// Mitsubishi GX Works2 project: Group 7 PLC   PLC: FX3G

// global labels: Global1
VAR_GLOBAL
  Emergency AT X005 : BOOL;
  PowerButton AT X007 : BOOL;
  PowerOn AT Y007 : BOOL;
  analog_input_1 AT D8280 : INT;
END_VAR
VAR_GLOBAL CONSTANT
  div_analog : REAL := 400.0;
  max_regular : REAL := 5.0;
  min_pinuk : REAL := 6.0;
END_VAR
VAR_GLOBAL
  pinuk AT M1 : BOOL;  (* fictive lamp that represent pinuk choise *)
  regular AT M2 : BOOL;  (* fictive lamp that represent regular choise *)
  RaspberryInput AT D1100 : REAL;
  LemonInput AT D1102 : REAL;
  StabilizerInput AT D1104 : REAL;
  GummyBearInput AT D1106 : REAL;
  RaspberryStock AT D1108 : REAL;
  LemonStock AT D1110 : REAL;
  StabilizerStock AT D1112 : REAL;
  GummyBearStock AT D1114 : REAL;
  RaspberryCoolingContainer AT D1116 : REAL;
  LemonCoolingContainer AT D1118 : REAL;
  MixingContainer AT D1120 : REAL;
  PackagesStorageContainer AT D1122 : REAL;
  analog_sample AT X001 : BOOL;
END_VAR
VAR_GLOBAL CONSTANT
  pinuk_gummy_pack : REAL := 70;
  pinuk_raspberry_pack : REAL := 385;
  pinuk_stabilizer_pack : REAL := 210;
END_VAR
VAR_GLOBAL
  out_of_stock AT M100 : BOOL;
END_VAR
VAR_GLOBAL CONSTANT
  regular_gummy_pack : REAL := 28;
  regular_lemon_pack : REAL := 455;
  regular_raspberry_pack : REAL := 280;
  regular_stabilizer_pack : REAL := 105;
  pinuk_lemon_pack : REAL := 665;
END_VAR
VAR_GLOBAL
  timer AT TC0 : BOOL;
END_VAR
VAR_GLOBAL CONSTANT
  flavors_interval : INT := 50;
END_VAR
VAR_GLOBAL
  flavors_timer AT TC0 : BOOL;
  flavors_timer_OUTPUT AT TS0 : BOOL;
  flavors_lamp AT Y000 : BOOL;
  start_cooling AT X002 : BOOL;
  finish_flavor_step AT M3 : BOOL;
END_VAR
VAR_GLOBAL CONSTANT
  Raspberry_pinuk_icecream : REAL := 560;
  Raspberry_regular_icecream : REAL := 350;
  lemon_pinuk_icecream : REAL := 700;
  lemon_regular_icecream : REAL := 490;
END_VAR
VAR_GLOBAL
  cooling_timer AT TC1 : BOOL;
  cooling_timer_OUTPUT AT TS1 : BOOL;
END_VAR
VAR_GLOBAL CONSTANT
  cooling_interval : INT := 80;
END_VAR
VAR_GLOBAL
  cooling_lamp AT Y002 : BOOL;
  temp_sensor AT X003 : BOOL;
  finish_cooling_step AT M4 : BOOL;
  flashing_fake_lamp AT M5 : BOOL;
  timer_flashing5 AT TC5 : BOOL;
END_VAR
VAR_GLOBAL CONSTANT
  flashing_timer : INT := 1;
END_VAR
VAR_GLOBAL
  outtimer_flashing5 AT TS5 : BOOL;
  lamp5 AT Y005 : BOOL;
  timer_flashing6 AT TC6 : BOOL;
  outtimer_flashing6 AT TS6 : BOOL;
  lamp6 AT Y006 : BOOL;
  timer_flashing56 AT TC56 : BOOL;
END_VAR
VAR_GLOBAL CONSTANT
  flashing_timer56 : INT := 30;
END_VAR
VAR_GLOBAL
  timer_flashing56_out AT TS56 : BOOL;
END_VAR
VAR_GLOBAL CONSTANT
  GummyBear_pinuk : REAL := 70;
  GummyBear_regular : REAL := 28;
  flashing_regular_timer56 : INT := 30;
  flashing_pinuk_timer56 : INT := 50;
END_VAR
VAR_GLOBAL
  timer_flashing2 AT TC2 : BOOL;
  timer_flashing3 AT TC3 : BOOL;
  timer_flashing2_out AT TS2 : BOOL;
  timer_flashing3_out AT TS3 : BOOL;
  packing_button AT X004 : BOOL;  (* fictive lamp that represent pinuk choise *)
  counter_x0 AT X000 : BOOL;
END_VAR
VAR_GLOBAL CONSTANT
  Sum_pack : INT := 7;
END_VAR
VAR_GLOBAL
  units_counter AT CC1 : BOOL;  (* fictive lamp that represent pinuk choise *)
  units_counter_OUT AT CS1 : BOOL;
  packing_lamp AT Y004 : BOOL;
END_VAR
VAR_GLOBAL CONSTANT
  value1 : INT := 1;
  value_is_1 : REAL := 1;
END_VAR
VAR_GLOBAL
  finish_iteretion AT M8 : BOOL;
  pinukM AT M10 : BOOL;  (* fictive lamp that represent pinuk choise *)
  regularM AT M20 : BOOL;  (* fictive lamp that represent pinuk choise *)
END_VAR
VAR_GLOBAL CONSTANT
  mul_analog : REAL := 40;
END_VAR
VAR_GLOBAL
  analog_output_1 AT D8282 : INT;
  fyuyu AT Y011 : BOOL;
  out_of_stock1 AT M102 : BOOL;
END_VAR

// task Task_01 (event TRUE, interval 0, priority 31): POU_01

PROGRAM POU_01
(* structured ladder/FBD written out as ST: instructions are called as NAME(EN, inputs, outputs); _pN, _eN, _tN stand for wires *)
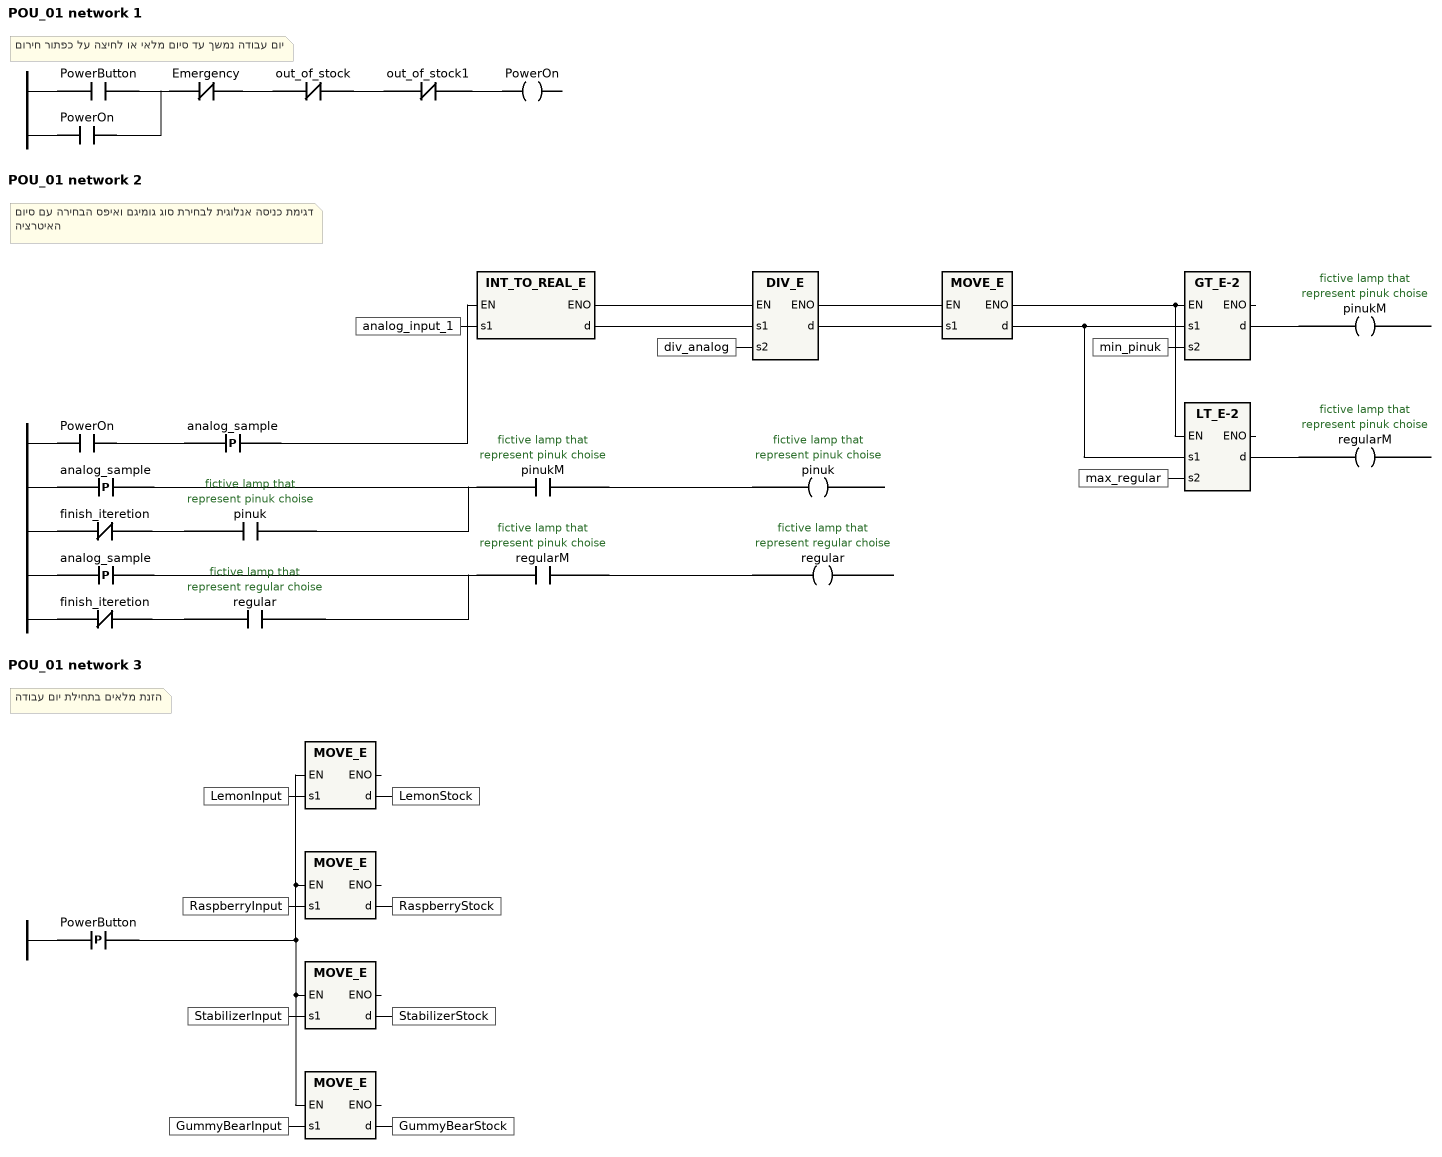
(* network 1 Start-Stop Day *)
(* יום עבודה נמשך עד סיום מלאי או לחיצה על כפתור חירום *)
PowerOn := (((PowerButton OR PowerOn) AND NOT Emergency) AND NOT out_of_stock) AND NOT out_of_stock1;
(* network 2 Analog Sample *)
(* דגימת כניסה אנלוגית לבחירת סוג גומיגם ואיפס הבחירה עם סיום האיטרציה *)
_e2 := INT_TO_REAL_E(PowerOn AND LDP(TRUE, analog_sample), analog_input_1, _t1);
_e4 := DIV_E(_e2, _t1, div_analog, _t3);
_e6 := MOVE_E(_e4, _t3, _t5);
GT_E(_e6, _t5, min_pinuk, _t7);
pinukM := _t7;
LT_E(_e6, _t5, max_regular, _t8);
regularM := _t8;
pinuk := (LDP(TRUE, analog_sample) OR (NOT finish_iteretion AND pinuk)) AND pinukM;
regular := (LDP(TRUE, analog_sample) OR (NOT finish_iteretion AND regular)) AND regularM;
(* network 3 Initialization Reg *)
(* הזנת מלאים בתחילת יום עבודה *)
_p1 := LDP(TRUE, PowerButton);
MOVE_E(_p1, LemonInput, LemonStock);
MOVE_E(_p1, RaspberryInput, RaspberryStock);
MOVE_E(_p1, StabilizerInput, StabilizerStock);
MOVE_E(_p1, GummyBearInput, GummyBearStock);
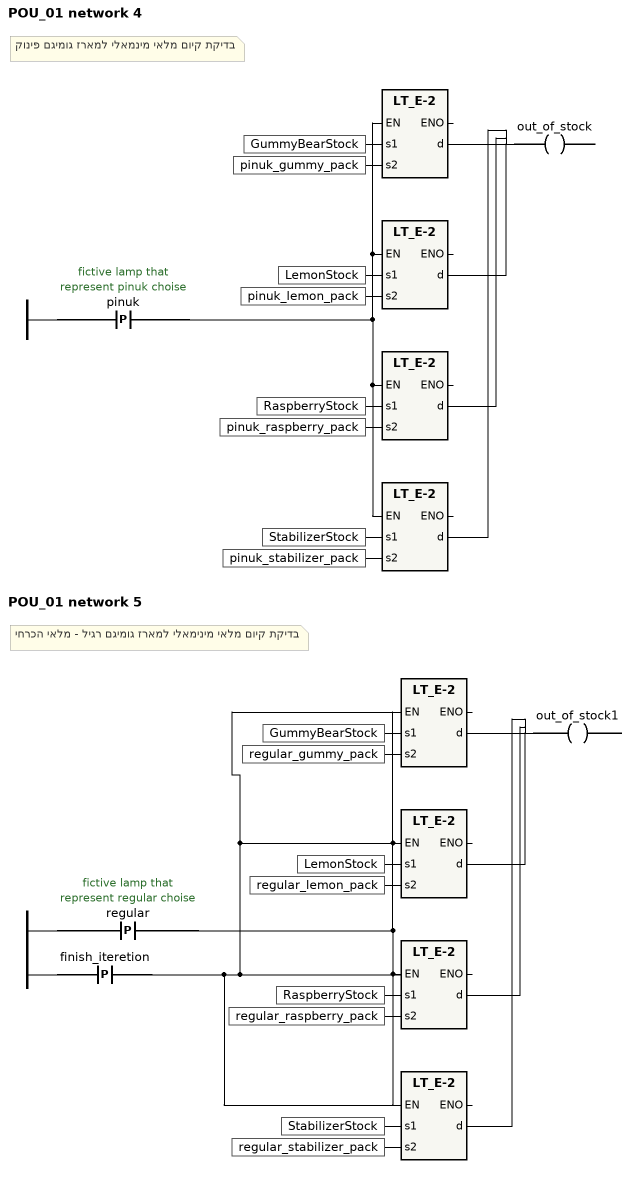
(* network 4 Pinuk Stock *)
(* בדיקת קיום מלאי מינמאלי למארז גומיגם פינוק *)
_p1 := LDP(TRUE, pinuk);
LT_E(_p1, GummyBearStock, pinuk_gummy_pack, _t2);
LT_E(_p1, LemonStock, pinuk_lemon_pack, _t3);
LT_E(_p1, RaspberryStock, pinuk_raspberry_pack, _t4);
LT_E(_p1, StabilizerStock, pinuk_stabilizer_pack, _t5);
out_of_stock := _t2 OR _t3 OR _t4 OR _t5;
(* network 5 Regular Stock *)
(* בדיקת קיום מלאי מינימאלי למארז גומיגם רגיל - מלאי הכרחי *)
_p1 := LDP(TRUE, regular) OR LDP(TRUE, finish_iteretion);
LT_E(_p1, GummyBearStock, regular_gummy_pack, _t2);
LT_E(_p1, LemonStock, regular_lemon_pack, _t3);
LT_E(_p1, RaspberryStock, regular_raspberry_pack, _t4);
LT_E(_p1, StabilizerStock, regular_stabilizer_pack, _t5);
out_of_stock1 := _t2 OR _t3 OR _t4 OR _t5;
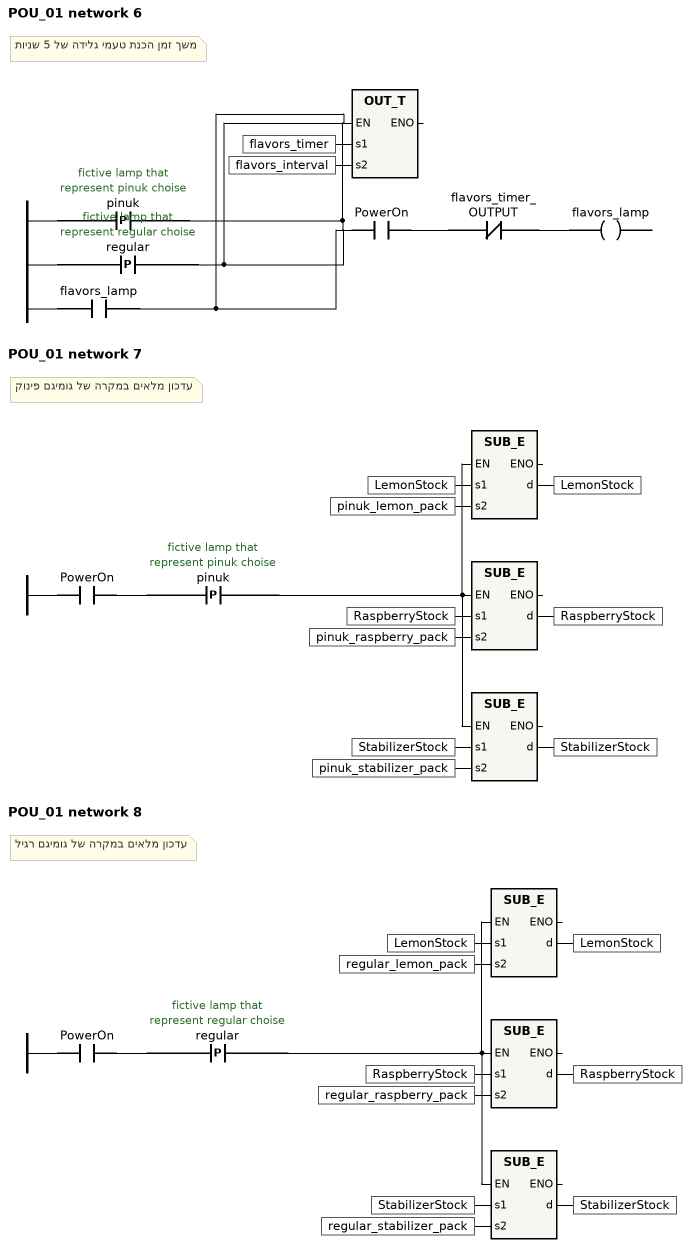
(* network 6 flavors_timer *)
(* משך זמן הכנת טעמי גלידה של 5 שניות *)
_p1 := LDP(TRUE, pinuk) OR LDP(TRUE, regular) OR flavors_lamp;
OUT_T(_p1, flavors_timer, flavors_interval);
flavors_lamp := _p1 AND PowerOn AND NOT flavors_timer_OUTPUT;
(* network 7 sub stocks pinuk *)
(* עדכון מלאים במקרה של גומיגם פינוק *)
_p1 := PowerOn AND LDP(TRUE, pinuk);
SUB_E(_p1, LemonStock, pinuk_lemon_pack, LemonStock);
SUB_E(_p1, RaspberryStock, pinuk_raspberry_pack, RaspberryStock);
SUB_E(_p1, StabilizerStock, pinuk_stabilizer_pack, StabilizerStock);
(* network 8 sub stocks regular *)
(* עדכון מלאים במקרה של גומיגם רגיל *)
_p1 := PowerOn AND LDP(TRUE, regular);
SUB_E(_p1, LemonStock, regular_lemon_pack, LemonStock);
SUB_E(_p1, RaspberryStock, regular_raspberry_pack, RaspberryStock);
SUB_E(_p1, StabilizerStock, regular_stabilizer_pack, StabilizerStock);
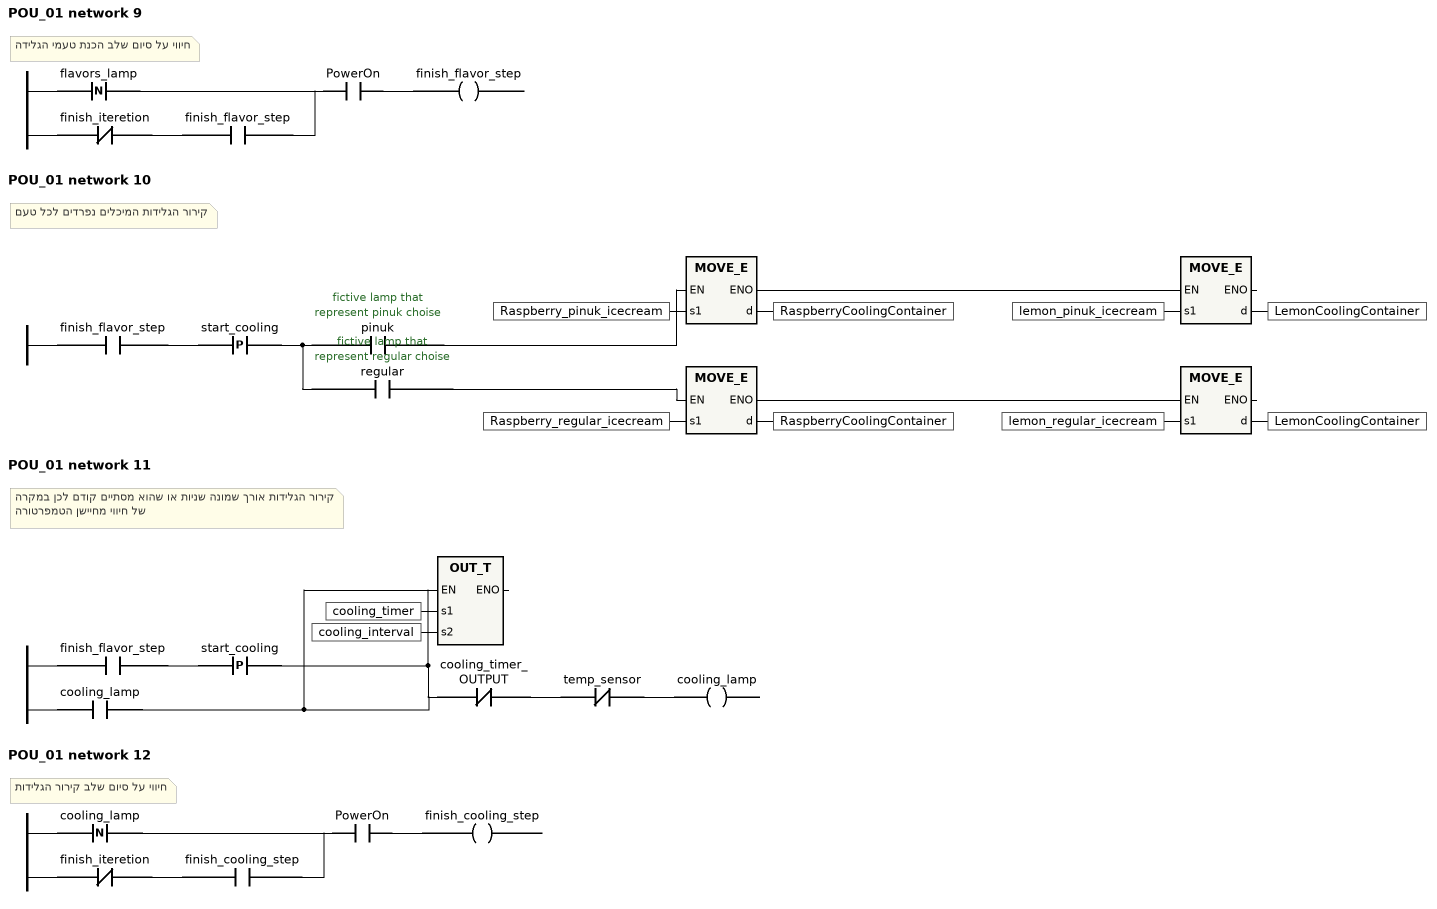
(* network 9 finish flavor step *)
(* חיווי על סיום שלב הכנת טעמי הגלידה *)
finish_flavor_step := (LDF(TRUE, flavors_lamp) OR (NOT finish_iteretion AND finish_flavor_step)) AND PowerOn;
(* network 10 cooling ice cream *)
(* קירור הגלידות המיכלים נפרדים לכל טעם *)
_p1 := finish_flavor_step AND LDP(TRUE, start_cooling);
_e2 := MOVE_E(_p1 AND pinuk, Raspberry_pinuk_icecream, RaspberryCoolingContainer);
MOVE_E(_e2, lemon_pinuk_icecream, LemonCoolingContainer);
_e3 := MOVE_E(_p1 AND regular, Raspberry_regular_icecream, RaspberryCoolingContainer);
MOVE_E(_e3, lemon_regular_icecream, LemonCoolingContainer);
(* network 11 cooling timer *)
(* קירור הגלידות אורך שמונה שניות או שהוא מסתיים קודם לכן במקרה של חיווי מחיישן הטמפרטורה *)
_p1 := (finish_flavor_step AND LDP(TRUE, start_cooling)) OR cooling_lamp;
OUT_T(_p1, cooling_timer, cooling_interval);
cooling_lamp := _p1 AND NOT cooling_timer_OUTPUT AND NOT temp_sensor;
(* network 12 finish cooling step *)
(* חיווי על סיום שלב קירור הגלידות *)
finish_cooling_step := (LDF(TRUE, cooling_lamp) OR (NOT finish_iteretion AND finish_cooling_step)) AND PowerOn;
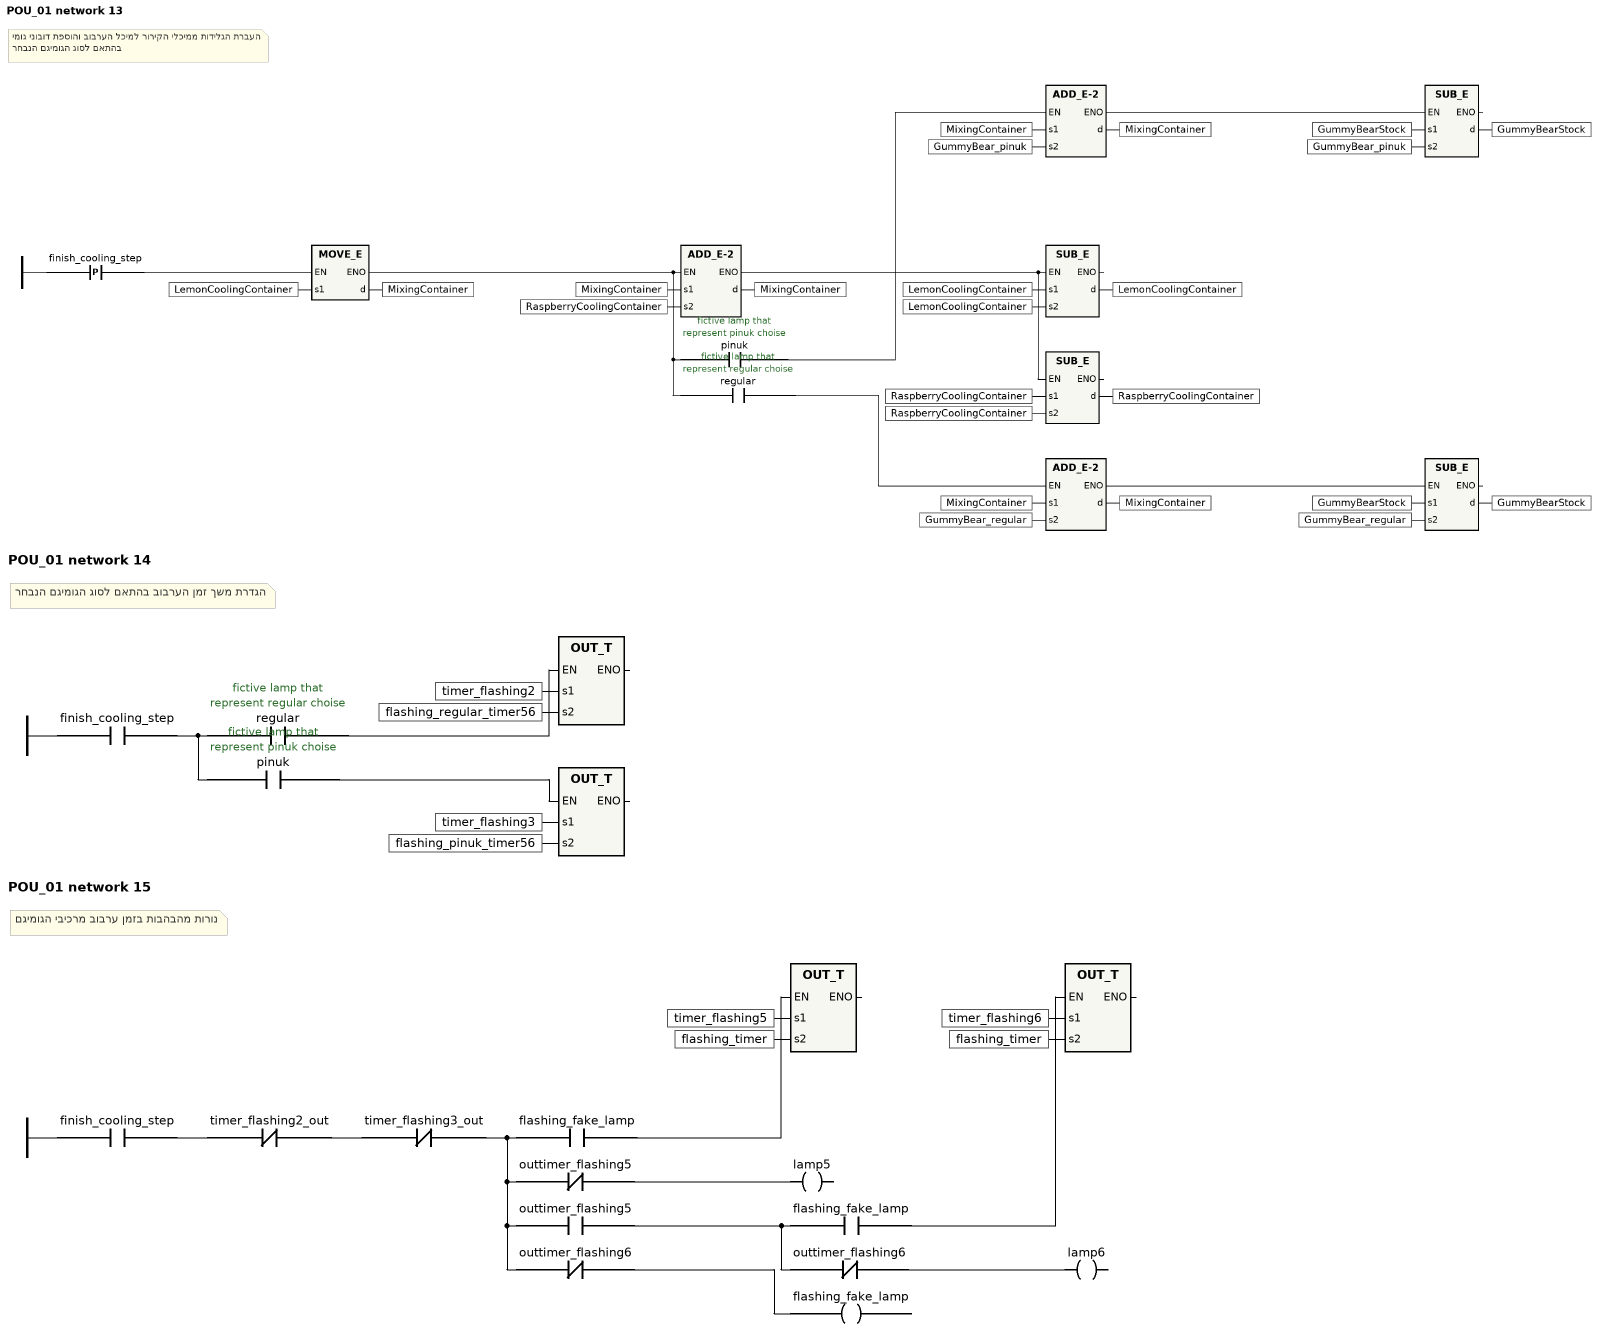
(* network 13 mixing *)
(* העברת הגלידות ממיכלי הקירור למיכל הערבוב והוספת דובוני גומי בהתאם לסוג הגומיגם הנבחר *)
_e1 := MOVE_E(LDP(TRUE, finish_cooling_step), LemonCoolingContainer, MixingContainer);
_e2 := ADD_E(_e1, MixingContainer, RaspberryCoolingContainer, MixingContainer);
SUB_E(_e2, LemonCoolingContainer, LemonCoolingContainer, LemonCoolingContainer);
SUB_E(_e2, RaspberryCoolingContainer, RaspberryCoolingContainer, RaspberryCoolingContainer);
_e3 := ADD_E(_e1 AND pinuk, MixingContainer, GummyBear_pinuk, MixingContainer);
SUB_E(_e3, GummyBearStock, GummyBear_pinuk, GummyBearStock);
_e4 := ADD_E(_e1 AND regular, MixingContainer, GummyBear_regular, MixingContainer);
SUB_E(_e4, GummyBearStock, GummyBear_regular, GummyBearStock);
(* network 14 flashing duration  *)
(* הגדרת משך זמן הערבוב בהתאם לסוג הגומיגם הנבחר *)
OUT_T(finish_cooling_step AND regular, timer_flashing2, flashing_regular_timer56);
OUT_T(finish_cooling_step AND pinuk, timer_flashing3, flashing_pinuk_timer56);
(* network 15 flashing lamps *)
(* נורות מהבהבות בזמן ערבוב מרכיבי הגומיגם *)
_p1 := finish_cooling_step AND NOT timer_flashing2_out AND NOT timer_flashing3_out;
OUT_T(_p1 AND flashing_fake_lamp, timer_flashing5, flashing_timer);
lamp5 := _p1 AND NOT outtimer_flashing5;
_p2 := _p1 AND outtimer_flashing5;
OUT_T(_p2 AND flashing_fake_lamp, timer_flashing6, flashing_timer);
lamp6 := _p2 AND NOT outtimer_flashing6;
flashing_fake_lamp := _p1 AND NOT outtimer_flashing6;
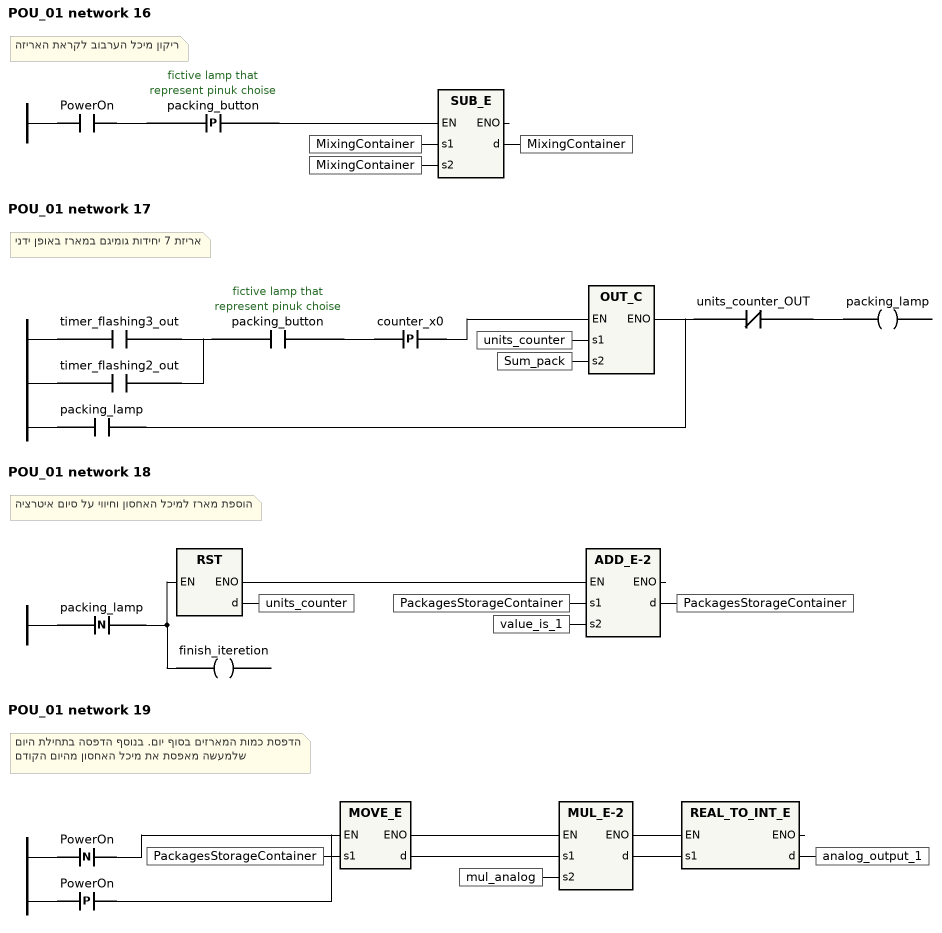
(* network 16 emptying mix cont *)
(* ריקון מיכל הערבוב לקראת האריזה *)
SUB_E(PowerOn AND LDP(TRUE, packing_button), MixingContainer, MixingContainer, MixingContainer);
(* network 17 packing process *)
(* אריזת 7 יחידות גומיגם במארז באופן ידני *)
_e1 := OUT_C(((timer_flashing3_out OR timer_flashing2_out) AND packing_button) AND LDP(TRUE, counter_x0), units_counter, Sum_pack);
packing_lamp := (_e1 OR packing_lamp) AND NOT units_counter_OUT;
(* network 18 7 units  *)
(* הוספת מארז למיכל האחסון וחיווי על סיום איטרציה *)
_p1 := LDF(TRUE, packing_lamp);
_e2 := RST(_p1, units_counter);
ADD_E(_e2, PackagesStorageContainer, value_is_1, PackagesStorageContainer);
finish_iteretion := _p1;
(* network 19 analog output *)
(* הדפסת כמות המארזים בסוף יום. בנוסף הדפסה בתחילת היום שלמעשה מאפסת את מיכל האחסון מהיום הקודם *)
_e2 := MOVE_E(LDF(TRUE, PowerOn) OR LDP(TRUE, PowerOn), PackagesStorageContainer, _t1);
_e4 := MUL_E(_e2, _t1, mul_analog, _t3);
REAL_TO_INT_E(_e4, _t3, analog_output_1);
END_PROGRAM
